// TIA Portal V20 export
VAR_GLOBAL   // PLC tag table "PLC_Centralizer"
   Digital_Input_0 AT %I0.0 : Bool;
   Digital_Input_1 AT %I0.1 : Bool;
   Digital_Input_2 AT %I0.2 : Bool;
   Digital_Input_3 AT %I0.3 : Bool;
   Digital_Input_4 AT %I0.4 : Bool;
   Digital_Input_5 AT %I0.5 : Bool;
   Digital_Input_6 AT %I0.6 : Bool;
   Digital_Input_7 AT %I0.7 : Bool;
   Digital_Input_8 AT %I1.0 : Bool;
   Digital_Input_9 AT %I1.1 : Bool;
   Digital_Input_10 AT %I1.2 : Bool;
   Digital_Input_11 AT %I1.3 : Bool;
   Digital_Input_12 AT %I1.4 : Bool;
   Digital_Input_13 AT %I1.5 : Bool;
   Analogic_Input_0 AT %IW64 : Int;
   Analogic_Input_1 AT %IW66 : Int;
   Digital_Output_0 AT %Q0.0 : Bool;
   Digital_Output_1 AT %Q0.1 : Bool;
   Digital_Output_2 AT %Q0.2 : Bool;
   Digital_Output_3 AT %Q0.3 : Bool;
   Digital_Output_4 AT %Q0.4 : Bool;
   Digital_Output_5 AT %Q0.5 : Bool;
   Digital_Output_6 AT %Q0.6 : Bool;
   Digital_Output_7 AT %Q0.7 : Bool;
   Digital_Output_8 AT %Q1.0 : Bool;
   Digital_Output_9 AT %Q1.1 : Bool;
   Clock_Byte AT %MB0 : Byte;
   Clock_10Hz AT %M0.0 : Bool;
   Clock_5Hz AT %M0.1 : Bool;
   "Clock_2.5Hz" AT %M0.2 : Bool;
   Clock_2Hz AT %M0.3 : Bool;
   "Clock_1.25Hz" AT %M0.4 : Bool;
   Clock_1Hz AT %M0.5 : Bool;
   "Clock_0.625Hz" AT %M0.6 : Bool;
   "Clock_0.5Hz" AT %M0.7 : Bool;
   System_Byte AT %MB1 : Byte;
   FirstScan AT %M1.0 : Bool;
   DiagStatusUpdate AT %M1.1 : Bool;
   AlwaysTRUE AT %M1.2 : Bool;
   AlwaysFALSE AT %M1.3 : Bool;
END_VAR
